{attribute 'qualified_only'}
{attribute 'strict'}
{attribute 'to_string'}
TYPE E_MESSAGE_BATCH :
(
	MSG_BATCH_NULL,
  MSG_BATCH_JOB_STARTED,
  MSG_BATCH_NEXT_IN_JOB,
  MSG_BATCH_JOB_DONE
)UINT;
END_TYPE

(* stored: Version 1.1.0.1
   DUT E_MESSAGE_BATCH: Id {5432bb4c-e002-46f8-8955-c6c287f6b579} *)
